{attribute 'qualified_only'}
{attribute 'strict'}
{attribute 'to_string'}
TYPE eMessageCategories :
(
	HardwareFailure := 0,
	TimeoutFailure := 1,
	MissingData := 2,
	LostConnection := 3,
	Undefined := 4,
	NotImplemented:=5,
	NotAllowed:=6
);
END_TYPE

(* stored: Version 1.1.0.1
   DUT eMessageCategories: Id {f686d474-7d27-4531-ac7a-80c2a5b3adc0} *)
